// TIA Portal V19 export
FUNCTION_BLOCK "TYPIC_C904_SF_PMP"   // FB133, FBD
TITLE = TYPIC_C904_SF_PMP: pomp
{ S7_Optimized_Access := 'TRUE' }
AUTHOR : OCOTECH
FAMILY : Typical
NAME : C904.803
// Logisch Object Besturing: C904.803
// 
// Het doel van deze subfunctie is om de algemene sturing en bediening vanuit 3B te voorzien van een pomp behorende tot de hoofdpompinstallatie.
// stored: MemoryReserve 10, SetENOAutomatically false
   VAR_INPUT
      CFG_PWR { ExternalAccessible := 'False'; ExternalVisible := 'False'; ExternalWritable := 'False'} : Real;   // Nominaal vermogen als pomp aangeschakeld
      STU_CMD_AUT { ExternalAccessible := 'False'; ExternalVisible := 'False'; ExternalWritable := 'False'} : USInt;   // Groepscommando: schakel in automatisch
      STU_ALG_LCK_SIG { ExternalAccessible := 'False'; ExternalVisible := 'False'; ExternalWritable := 'False'} : USInt;   // Onderdruk alarmen
      STU_ENE_VGV_AAN { ExternalAccessible := 'False'; ExternalVisible := 'False'; ExternalWritable := 'False'} : USInt;   // Vrijgeven of verhinderen bijschakelen energieverbruikers (verlichting / ventilatie)
   END_VAR
   VAR_OUTPUT
      VAR_PMP { ExternalAccessible := 'False'; ExternalVisible := 'False'; ExternalWritable := 'False'} : "C904_VAR_PMP_TYPIC";   // Struct met alle variabelen van de pomp
      STU_IF_PMP { ExternalAccessible := 'False'; ExternalVisible := 'False'; ExternalWritable := 'False'} : "C904_STU_IF_PMP_TYPIC";   // Struct met alle sturingen naar de functie (IF) in de interne sturing van de pomp
   END_VAR
   VAR_IN_OUT
      STU_PMP_CMD : USInt;   // Sturing pomp (vanuit de basisfunctie)
      VAR_IF_PMP : "C904_VAR_IF_PMP_TYPIC";   // Struct met alle variabelen van de pomp, ontvangen vanuit de interne sturing
   END_VAR
   VAR
      BED : Struct   // Bedieningen
         ALG : Struct   // Gewenste stand
            X : "UDT_BED_ALG";
            KNOP { S7_SetPoint := 'True'} : Array[0..2] of "UDT_BED_KNOP";
         END_STRUCT;
         BST : Struct   // Bestuurbaarheid
            X : "UDT_BED_ALG";
            KNOP { S7_SetPoint := 'True'} : Array[0..1] of "UDT_BED_KNOP";
         END_STRUCT;
         RES : Struct   // Reset storingen
            X : "UDT_BED_ALG";
            KNOP { S7_SetPoint := 'True'} : Array[0..0] of "UDT_BED_KNOP";
         END_STRUCT;
      END_STRUCT;
      BED_ALG { ExternalWritable := 'False'} : "TYPIC_HF_BED_ALG_KNOP";   // Gewenste stand
      BED_BST { ExternalWritable := 'False'} : "TYPIC_HF_BED_ALG_KNOP";   // Bestuurbaarheid
      BED_RES { ExternalWritable := 'False'} : "TYPIC_HF_BED_ALG_KNOP";   // Reset storingen
      SIG { ExternalWritable := 'False'} : Struct   // Signaleringen
         AA01 : Bool;   // Pomp niet bestuurbaar
         AA02 : Bool;   // Storing algemeen
         A001 : Bool;   // Beveiliging aangesproken
         A002 : Bool;   // Storing van de motorbeveiliging van de pomp
         A003 : Bool;   // Storing motorlade
         A004 : Bool;   // Te hoge temperatuur in de motorwikkelingen
         A005 : Bool;   // Fout stroommeting fase 1
         A006 : Bool;   // Fout stroommeting fase 2
         A007 : Bool;   // Fout stroommeting fase 3
         A008 : Bool;   // Droogloop beveiliging actief: LLW vlotter bovenwater
         A009 : Bool;   // Lekdetectie pomp
         A010 : Bool;   // Motorlade uitgeschakeld
         A011 : Bool;   // Motorlade in test
         A012 : Bool;   // Motorlade uitgereden
         AT01 : Bool;   // Discordantie motor: terugmelding niet ontvangen
         AT02 : Bool;   // Discordantie motor: terugmelding blijft aanwezig
         M001 : Bool;   // Werkschakelaar uitgeschakeld
         M002 : Bool;   // Melding: Pomp heeft te lang niet gedraaid. Periodiek onderhoud nodig
      END_STRUCT;
      VAR { ExternalWritable := 'False'} : Struct   // Variabelen
         TYD_TOT_AAN_UUR : USInt;   // Totaal aantal draaiuren
         ENE_MWA1 : USInt;   // Stroommeting fase 1
         ENE_MWA2 : USInt;   // Stroommeting fase 2
         ENE_MWA3 : USInt;   // Stroommeting fase 3
         RNB : USInt;   // Reden niet bestuurbaar
         AUT : USInt;   // Beveiliging aangesproken
         VGV_SIG_VOP : Bool;   // TRUE = Signaleringen vrijgegeven voor verkeersoperator FALSE = Onderdrukt
         STS : USInt;   // Status van de pomp
         BMO : USInt;   // Bedieningsmode
         BST { ExternalAccessible := 'False'; ExternalVisible := 'False'} : USInt;   // Bestuurbaarheid
         LLW { ExternalAccessible := 'False'; ExternalVisible := 'False'} : USInt;   // Vlotter droogloopbewaking
         PWR { ExternalAccessible := 'False'; ExternalVisible := 'False'} : Real;   // Actueel vermogen van de pomp
         TYD_TOT_AAN { ExternalAccessible := 'False'; ExternalVisible := 'False'} : USInt;   // Totaal aantal draaiuren
         TYD_AAN { ExternalAccessible := 'False'; ExternalVisible := 'False'} : USInt;   // Tijdsduur dat pomp aangeschakeld is
         TYD_UIT { ExternalAccessible := 'False'; ExternalVisible := 'False'} : USInt;   // Tijdsduur dat pomp uitgeschakeld is
      END_STRUCT;
      HF_BST_OBS { ExternalAccessible := 'False'; ExternalVisible := 'False'; ExternalWritable := 'False'} : "TYPIC_HF_BST_OBS";   // Hulp functie besturing
   END_VAR
   // // BED.ALG.KNOP[0] : AUTO
   // // BED.ALG.KNOP[1] : Aan
   // // BED.ALG.KNOP[2] : Uit
   // // BED.BST.KNOP[0] : InDienst
   // // BED.BST.KNOP[1] : UitDienst
   // // BED.RES.KNOP[0] : Reset
BEGIN

REGION Network 1: START
END_REGION

REGION Network 2: +++ Bedieningen +++
   // Vrijgave en verwerking van de bedieningen (centrale en lokale bediening). De bedienwaardes worden daarna in de verdere deelfunctionaliteiten gebruikt.
END_REGION

REGION Network 3: Knoppen BED_ALG(Gewenste stand)
   // Waardes en vrijge van de knoppen BED_ALG
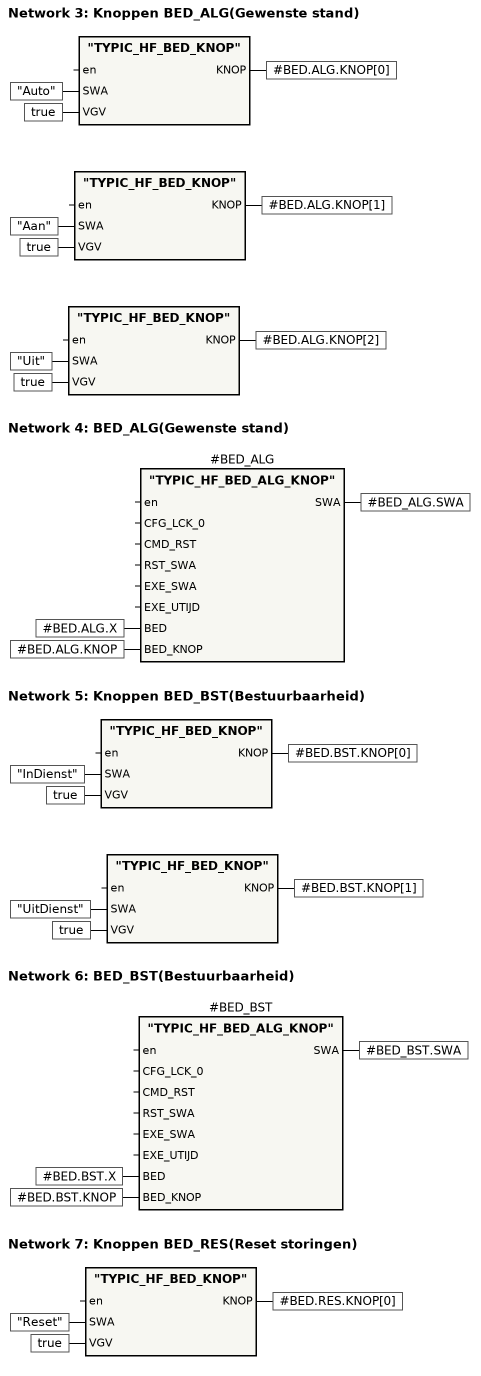
   "TYPIC_HF_BED_KNOP"(SWA := "Auto", VGV := true, KNOP => #BED.ALG.KNOP[0]);
   "TYPIC_HF_BED_KNOP"(SWA := "Aan", VGV := true, KNOP => #BED.ALG.KNOP[1]);
   "TYPIC_HF_BED_KNOP"(SWA := "Uit", VGV := true, KNOP => #BED.ALG.KNOP[2]);
END_REGION

REGION Network 4: BED_ALG(Gewenste stand)
   // Verwerking BED_ALG
   #BED_ALG(BED := #BED.ALG.X, BED_KNOP := #BED.ALG.KNOP, SWA => #BED_ALG.SWA);   // "TYPIC_HF_BED_ALG_KNOP"
END_REGION

REGION Network 5: Knoppen BED_BST(Bestuurbaarheid)
   // Waardes en vrijge van de knoppen BED_BST
   "TYPIC_HF_BED_KNOP"(SWA := "InDienst", VGV := true, KNOP => #BED.BST.KNOP[0]);
   "TYPIC_HF_BED_KNOP"(SWA := "UitDienst", VGV := true, KNOP => #BED.BST.KNOP[1]);
END_REGION

REGION Network 6: BED_BST(Bestuurbaarheid)
   // Verwerking BED_BST
   #BED_BST(BED := #BED.BST.X, BED_KNOP := #BED.BST.KNOP, SWA => #BED_BST.SWA);   // "TYPIC_HF_BED_ALG_KNOP"
END_REGION

REGION Network 7: Knoppen BED_RES(Reset storingen)
   // Waardes en vrijge van de knoppen BED_RES
   "TYPIC_HF_BED_KNOP"(SWA := "Reset", VGV := true, KNOP => #BED.RES.KNOP[0]);
END_REGION

REGION Network 8: BED_RES(Reset storingen)
   // Verwerking BED_RES
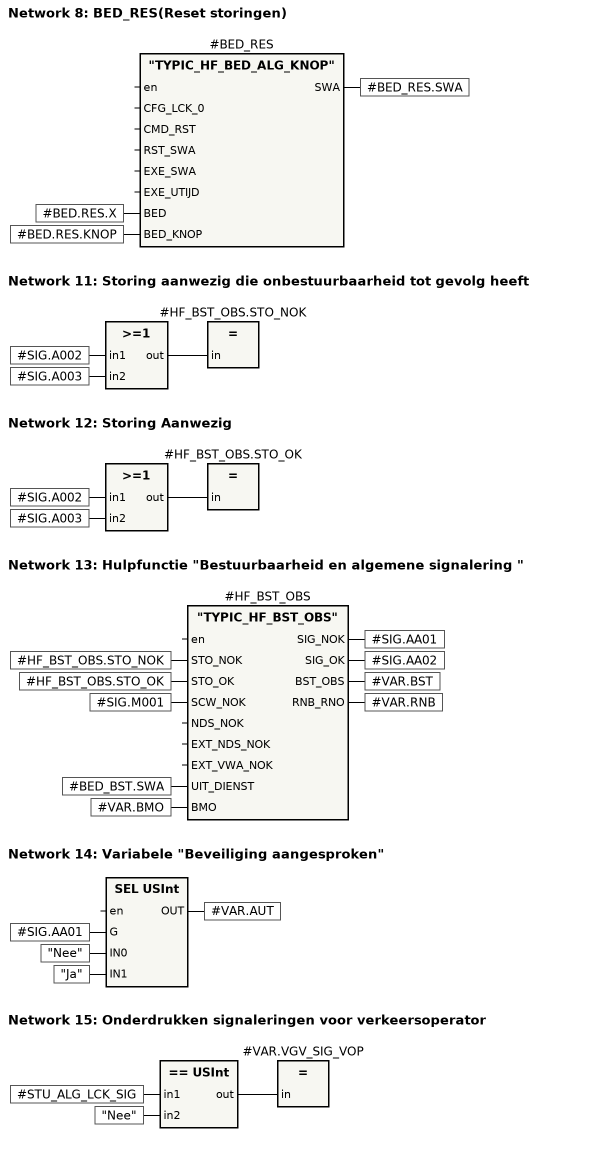
   #BED_RES(BED := #BED.RES.X, BED_KNOP := #BED.RES.KNOP, SWA => #BED_RES.SWA);   // "TYPIC_HF_BED_ALG_KNOP"
END_REGION

REGION Network 9: +++ Bepalen bedieningsmode +++
   // Bedieningsmode (Auto / Manueel / Hand) bepalen.
END_REGION

REGION Network 10: +++ Signaleringen en bestuurbaarheid +++
   // Aanmaken signaleringen, bepalen bestuurbaarheid (bestuurbaar / niet bestuurbaar) en bepalen reden van niet bestuurbaarheid.
END_REGION

REGION Network 11: Storing aanwezig die onbestuurbaarheid tot gevolg heeft
   // OR-verknoping van alle storingen om input STO_BST_NOK van de hulpfunctie "Bestuurbaarheid en algemene signlaring"
   #HF_BST_OBS.STO_NOK := #SIG.A002 OR #SIG.A003;
END_REGION

REGION Network 12: Storing Aanwezig
   // OR-verknoping van alle storingen om input STO_BST_OK van de hulpfunctie "Bestuurbaarheid en algemene signlaring"
   #HF_BST_OBS.STO_OK := #SIG.A002 OR #SIG.A003;
END_REGION

REGION Network 13: Hulpfunctie "Bestuurbaarheid en algemene signalering "
   // Bepalen variabele "bestuurbaarheid" en "reden niet bestuurbaar", Signaleringen "bestuurbaarheid" en "algmene storing".
   #HF_BST_OBS(STO_NOK := #HF_BST_OBS.STO_NOK,   // "TYPIC_HF_BST_OBS"
               STO_OK := #HF_BST_OBS.STO_OK,
               SCW_NOK := #SIG.M001,
               UIT_DIENST := #BED_BST.SWA,
               BMO := #VAR.BMO,
               SIG_NOK => #SIG.AA01,
               SIG_OK => #SIG.AA02,
               BST_OBS => #VAR.BST,
               RNB_RNO => #VAR.RNB);
END_REGION

REGION Network 14: Variabele "Beveiliging aangesproken"
   // De variabele VAR_AUT geef aan of er een beveilliging aangesproken is. Deze variabele laat toe dat de verkeersoperator op SCADA kan zien of er een beveilliging aangesproken is voor deze component.
   #VAR.AUT := SEL(G := #SIG.AA01, IN0 := "Nee", IN1 := "Ja");
END_REGION

REGION Network 15: Onderdrukken signaleringen voor verkeersoperator
   // Via de variabele VGV_SIG_VOP wordt aan IRIS SCADA doorgegeven of signaleringen (bestemd voor de verkeersoperator) van de deze functie zichtbaar (of onderdrukt) moeten zijn.
   #VAR.VGV_SIG_VOP := #STU_ALG_LCK_SIG = "Nee";
END_REGION

REGION Network 16: +++ Bepalen status en actueel vermogen +++
   // Status (Aan / Uit) en actueel verbruikt vermogen bepalen.
END_REGION

REGION Network 17: +++ Draaiuren en fasestromen +++
   // Totaal aantal draaiuren, momentaan aantal draaiuren (actueel aantal uren dat pomp draait / actueel aantal uren dat pomp stilstaat) en fasestromen bepalen.
END_REGION

REGION Network 18: +++ Sturingen +++
   // Commandos naar de interne sturing van de pomp uitsturen.
END_REGION

REGION Network 19 (SCL): EINDE
   // Variabelen van intern scada rakvlak naar outputs copieren
   #VAR_PMP.STS := #VAR.STS;
   #VAR_PMP.BMO := #VAR.BMO;
   #VAR_PMP.BST := #VAR.BST;
   #VAR_PMP.LLW := #VAR.LLW;
   #VAR_PMP.PWR := #VAR.PWR;
   #VAR_PMP.TYD_TOT_AAN := #VAR.TYD_TOT_AAN;
   #VAR_PMP.TYD_AAN := #VAR.TYD_AAN;
   #VAR_PMP.TYD_UIT := #VAR.TYD_UIT;
END_REGION
END_FUNCTION_BLOCK
